TYPE ST_BatchData :
STRUCT
	Batch		: STRING(100);
	Parameter	: STRING(100);
	Value		: STRING(100);
END_STRUCT
END_TYPE

(* stored: Version 1.1.0.1, ProductVersion 3.1.4024.12
   DUT ST_BatchData: Id {16d0d617-414a-4621-8d09-2ffe509f5573} *)
